{attribute 'qualified_only'}
{attribute 'strict'}
{attribute 'to_string'}
TYPE Food :
(
    Nothing,
    Carrot,
    Cabbage,
    Broccoli,
    Peas,
    Tofu,
    Humous,
    LentilCurry
);
END_TYPE

(* stored: Version 1.1.0.1, ProductVersion 3.1.4024.13
   DUT Food: Id {8b460533-974d-4a5f-a6e6-5d277f2da8e4} *)
